// IO/CtrlInput
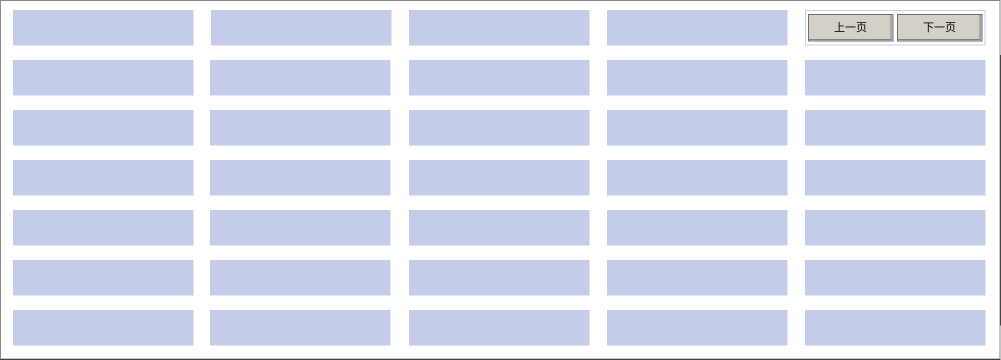
VISUALIZATION CtrlInput  // 1001x360
VAR_INPUT
	In:						POINTER TO BOOL;
	SizeIn:					DINT;
END_VAR
VAR
	_pageCount:				INT;
	_index:					INT;
END_VAR
    RoundedRectangle (0,0 1000x115)
    RoundedRectangle (0,245 1000x115)
    Rectangle (0,71 1000x240)
    Line (1000,55) (1000,325)
    Line (0,65) (0,312)
    RoundedRectangle (13,10 180x35), colour toggle: In[_index], invisible if: SizeIn<=_index, text list: 'InputText', text index: _index
    RoundedRectangle (211,10 180x35), colour toggle: In[1+_index], invisible if: SizeIn<= 1+_index, text list: 'InputText', text index: 1+_index
    RoundedRectangle (409,10 180x35), colour toggle: In[2+_index], invisible if: SizeIn<= 2+_index, text list: 'InputText', text index: 2+_index
    RoundedRectangle (607,10 180x35), colour toggle: In[3+_index], invisible if: SizeIn<=3+_index, text list: 'InputText', text index: 3+_index
    RoundedRectangle (805,10 180x35)
    Button (808,14 85x27), "上一页"
        OnMouseClick: execute {
            IF _index-34>=0 THEN
            	_index:=_index-34;
            END_IF
        }
    Button (897,14 85x27), "下一页"
        OnMouseClick: execute {
            IF SizeIn>_index+34 THEN
            	_index:=_index+34;
            END_IF
        }
    RoundedRectangle (13,60 180x35), colour toggle: In[_index+4], invisible if: SizeIn<=_index+4, text list: 'InputText', text index: _index+4
    RoundedRectangle (210,60 180x35), colour toggle: In[_index+5], invisible if: SizeIn<=_index+5, text list: 'InputText', text index: _index+5
    RoundedRectangle (409,60 180x35), colour toggle: In[_index+6], invisible if: SizeIn<=_index+6, text list: 'InputText', text index: _index+6
    RoundedRectangle (607,60 180x35), colour toggle: In[_index+7], invisible if: SizeIn<=_index+7, text list: 'InputText', text index: _index+7
    RoundedRectangle (805,60 180x35), colour toggle: In[_index+8], invisible if: SizeIn<=_index+8, text list: 'InputText', text index: _index+8
    RoundedRectangle (13,110 180x35), colour toggle: In[_index+9], invisible if: SizeIn<=_index+9, text list: 'InputText', text index: _index+9
    RoundedRectangle (210,110 180x35), colour toggle: In[_index+10], invisible if: SizeIn<=_index+10, text list: 'InputText', text index: _index+10
    RoundedRectangle (409,110 180x35), colour toggle: In[_index+11], invisible if: SizeIn<=_index+11, text list: 'InputText', text index: _index+11
    RoundedRectangle (607,110 180x35), colour toggle: In[_index+12], invisible if: SizeIn<=_index+12, text list: 'InputText', text index: _index+12
    RoundedRectangle (805,110 180x35), colour toggle: In[_index+13], invisible if: SizeIn<=_index+13, text list: 'InputText', text index: _index+13
    RoundedRectangle (13,160 180x35), colour toggle: In[_index+14], invisible if: SizeIn<=_index+14, text list: 'InputText', text index: _index+14
    RoundedRectangle (210,160 180x35), colour toggle: In[_index+15], invisible if: SizeIn<=_index+15, text list: 'InputText', text index: _index+15
    RoundedRectangle (409,160 180x35), colour toggle: In[_index+16], invisible if: SizeIn<=_index+16, text list: 'InputText', text index: _index+16
    RoundedRectangle (607,160 180x35), colour toggle: In[_index+17], invisible if: SizeIn<=_index+17, text list: 'InputText', text index: _index+17
    RoundedRectangle (805,160 180x35), colour toggle: In[_index+18], invisible if: SizeIn<=_index+18, text list: 'InputText', text index: _index+18
    RoundedRectangle (13,210 180x35), colour toggle: In[_index+19], invisible if: SizeIn<=_index+19, text list: 'InputText', text index: _index+19
    RoundedRectangle (210,210 180x35), colour toggle: In[_index+20], invisible if: SizeIn<=_index+20, text list: 'InputText', text index: _index+20
    RoundedRectangle (409,210 180x35), colour toggle: In[_index+21], invisible if: SizeIn<=_index+21, text list: 'InputText', text index: _index+21
    RoundedRectangle (607,210 180x35), colour toggle: In[_index+22], invisible if: SizeIn<=_index+22, text list: 'InputText', text index: _index+22
    RoundedRectangle (805,210 180x35), colour toggle: In[_index+23], invisible if: SizeIn<=_index+23, text list: 'InputText', text index: _index+23
    RoundedRectangle (13,260 180x35), colour toggle: In[_index+24], invisible if: SizeIn<=_index+24, text list: 'InputText', text index: _index+24
    RoundedRectangle (409,260 180x35), colour toggle: In[_index+26], invisible if: SizeIn<=_index+26, text list: 'InputText', text index: _index+26
    RoundedRectangle (210,260 180x35), colour toggle: In[_index+25], invisible if: SizeIn<=_index+25, text list: 'InputText', text index: _index+25
    RoundedRectangle (607,260 180x35), colour toggle: In[_index+27], invisible if: SizeIn<=_index+27, text list: 'InputText', text index: _index+27
    RoundedRectangle (805,260 180x35), colour toggle: In[_index+28], invisible if: SizeIn<=_index+28, text list: 'InputText', text index: _index+28
    RoundedRectangle (13,310 180x35), colour toggle: In[_index+29], invisible if: SizeIn<=_index+29, text list: 'InputText', text index: _index+29
    RoundedRectangle (210,310 180x35), colour toggle: In[_index+30], invisible if: SizeIn<=_index+30, text list: 'InputText', text index: _index+30
    RoundedRectangle (409,310 180x35), colour toggle: In[_index+31], invisible if: SizeIn<=_index+31, text list: 'InputText', text index: _index+31
    RoundedRectangle (607,310 180x35), colour toggle: In[_index+32], invisible if: SizeIn<=_index+32, text list: 'InputText', text index: _index+32
    RoundedRectangle (805,310 180x35), colour toggle: In[_index+33], invisible if: SizeIn<=_index+33, text list: 'InputText', text index: _index+33
END_VISUALIZATION

// IO/CtrlOutput
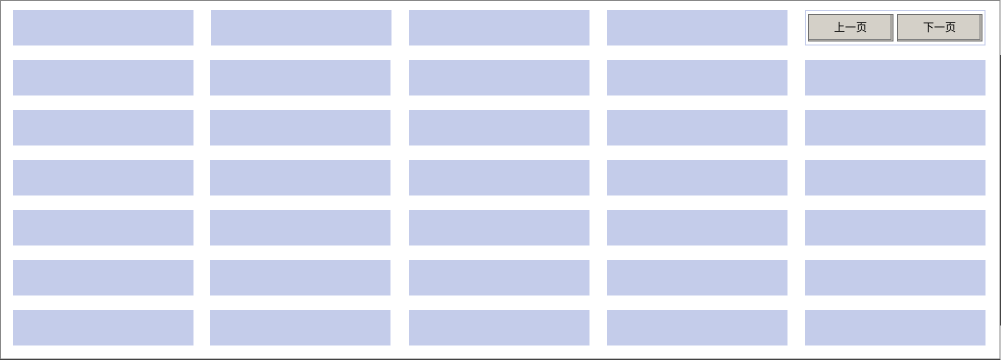
VISUALIZATION CtrlOutput  // 1001x360
VAR_INPUT
	In:						POINTER TO BOOL;
	SizeIn:					DINT;
	System:					REFERENCE TO ST_System;
END_VAR
VAR
	_pageCount:				INT;
	_index:					INT;
END_VAR
    RoundedRectangle (0,0 1000x115)
    RoundedRectangle (0,245 1000x115)
    Rectangle (0,71 1000x240)
    Line (1000,55) (1000,325)
    Line (0,65) (0,312)
    RoundedRectangle (13,10 180x35), colour toggle: In[_index], invisible if: SizeIn<=_index, text list: 'OutputText', text index: _index
        OnMouseClick: execute {
            IF System.stMode.bSetting AND SizeIn>_index THEN
            	In[_index]:=NOT In[_index];
            END_IF;
        }
    RoundedRectangle (211,10 180x35), colour toggle: In[1+_index], invisible if: SizeIn<= 1+_index, text list: 'OutputText', text index: 1+_index
        OnMouseClick: execute {
            IF System.stMode.bSetting AND SizeIn>_index+1 THEN
            	In[_index+1]:=NOT In[_index+1];
            END_IF;
        }
    RoundedRectangle (409,10 180x35), colour toggle: In[2+_index], invisible if: SizeIn<= 2+_index, text list: 'OutputText', text index: 2+_index
        OnMouseClick: execute {
            IF System.stMode.bSetting AND SizeIn>_index+2 THEN
            	In[_index+2]:=NOT In[_index+2];
            END_IF;
        }
    RoundedRectangle (607,10 180x35), colour toggle: In[3+_index], invisible if: SizeIn<=3+_index, text list: 'OutputText', text index: 3+_index
        OnMouseClick: execute {
            IF System.stMode.bSetting AND SizeIn>_index+3 THEN
            	In[_index+3]:=NOT In[_index+3];
            END_IF;
        }
    RoundedRectangle (805,10 180x35)
    RoundedRectangle (13,60 180x35), colour toggle: In[_index+4], invisible if: SizeIn<=_index+4, text list: 'OutputText', text index: _index+4
        OnMouseClick: execute {
            IF System.stMode.bSetting AND SizeIn>_index+4 THEN
            	In[_index+4]:=NOT In[_index+4];
            END_IF;
        }
    RoundedRectangle (210,60 180x35), colour toggle: In[_index+5], invisible if: SizeIn<=_index+5, text list: 'OutputText', text index: _index+5
        OnMouseClick: execute {
            IF System.stMode.bSetting AND SizeIn>_index+5 THEN
            	In[_index+5]:=NOT In[_index+5];
            END_IF;
        }
    RoundedRectangle (409,60 180x35), colour toggle: In[_index+6], invisible if: SizeIn<=_index+6, text list: 'OutputText', text index: _index+6
        OnMouseClick: execute {
            IF System.stMode.bSetting AND SizeIn>_index+6 THEN
            	In[_index+6]:=NOT In[_index+6];
            END_IF;
        }
    RoundedRectangle (607,60 180x35), colour toggle: In[_index+7], invisible if: SizeIn<=_index+7, text list: 'OutputText', text index: _index+7
        OnMouseClick: execute {
            IF System.stMode.bSetting AND SizeIn>_index+7 THEN
            	In[_index+7]:=NOT In[_index+7];
            END_IF;
        }
    RoundedRectangle (805,60 180x35), colour toggle: In[_index+8], invisible if: SizeIn<=_index+8, text list: 'OutputText', text index: _index+8
        OnMouseClick: execute {
            IF System.stMode.bSetting AND SizeIn>_index+8 THEN
            	In[_index+8]:=NOT In[_index+8];
            END_IF;
        }
    RoundedRectangle (13,110 180x35), colour toggle: In[_index+9], invisible if: SizeIn<=_index+9, text list: 'OutputText', text index: _index+9
        OnMouseClick: execute {
            IF System.stMode.bSetting AND SizeIn>_index+9 THEN
            	In[_index+9]:=NOT In[_index+9];
            END_IF;
        }
    RoundedRectangle (210,110 180x35), colour toggle: In[_index+10], invisible if: SizeIn<=_index+10, text list: 'OutputText', text index: _index+10
        OnMouseClick: execute {
            IF System.stMode.bSetting AND SizeIn>_index+10 THEN
            	In[_index+10]:=NOT In[_index+10];
            END_IF;
        }
    RoundedRectangle (409,110 180x35), colour toggle: In[_index+11], invisible if: SizeIn<=_index+11, text list: 'OutputText', text index: _index+11
        OnMouseClick: execute {
            IF System.stMode.bSetting AND SizeIn>_index+11 THEN
            	In[_index+11]:=NOT In[_index+11];
            END_IF;
        }
    RoundedRectangle (607,110 180x35), colour toggle: In[_index+12], invisible if: SizeIn<=_index+12, text list: 'OutputText', text index: _index+12
        OnMouseClick: execute {
            IF System.stMode.bSetting AND SizeIn>_index+12 THEN
            	In[_index+12]:=NOT In[_index+12];
            END_IF;
        }
    RoundedRectangle (805,110 180x35), colour toggle: In[_index+13], invisible if: SizeIn<=_index+13, text list: 'OutputText', text index: _index+13
        OnMouseClick: execute {
            IF System.stMode.bSetting AND SizeIn>_index+13 THEN
            	In[_index+13]:=NOT In[_index+13];
            END_IF;
        }
    RoundedRectangle (13,160 180x35), colour toggle: In[_index+14], invisible if: SizeIn<=_index+14, text list: 'OutputText', text index: _index+14
        OnMouseClick: execute {
            IF System.stMode.bSetting AND SizeIn>_index+14 THEN
            	In[_index+14]:=NOT In[_index+14];
            END_IF;
        }
    RoundedRectangle (210,160 180x35), colour toggle: In[_index+15], invisible if: SizeIn<=_index+15, text list: 'OutputText', text index: _index+15
        OnMouseClick: execute {
            IF System.stMode.bSetting AND SizeIn>_index+15 THEN
            	In[_index+15]:=NOT In[_index+15];
            END_IF;
        }
    RoundedRectangle (409,160 180x35), colour toggle: In[_index+16], invisible if: SizeIn<=_index+16, text list: 'OutputText', text index: _index+16
        OnMouseClick: execute {
            IF System.stMode.bSetting AND SizeIn>_index+16 THEN
            	In[_index+16]:=NOT In[_index+16];
            END_IF;
        }
    RoundedRectangle (607,160 180x35), colour toggle: In[_index+17], invisible if: SizeIn<=_index+17, text list: 'OutputText', text index: _index+17
        OnMouseClick: execute {
            IF System.stMode.bSetting AND SizeIn>_index+17 THEN
            	In[_index+17]:=NOT In[_index+17];
            END_IF;
        }
    RoundedRectangle (805,160 180x35), colour toggle: In[_index+18], invisible if: SizeIn<=_index+18, text list: 'OutputText', text index: _index+18
        OnMouseClick: execute {
            IF System.stMode.bSetting AND SizeIn>_index+18 THEN
            	In[_index+18]:=NOT In[_index+18];
            END_IF;
        }
    RoundedRectangle (13,210 180x35), colour toggle: In[_index+19], invisible if: SizeIn<=_index+19, text list: 'OutputText', text index: _index+19
        OnMouseClick: execute {
            IF System.stMode.bSetting AND SizeIn>_index+19 THEN
            	In[_index+19]:=NOT In[_index+19];
            END_IF;
        }
    RoundedRectangle (210,210 180x35), colour toggle: In[_index+20], invisible if: SizeIn<=_index+20, text list: 'OutputText', text index: _index+20
        OnMouseClick: execute {
            IF System.stMode.bSetting AND SizeIn>_index+20 THEN
            	In[_index+20]:=NOT In[_index+20];
            END_IF;
        }
    RoundedRectangle (409,210 180x35), colour toggle: In[_index+21], invisible if: SizeIn<=_index+21, text list: 'OutputText', text index: _index+21
        OnMouseClick: execute {
            IF System.stMode.bSetting AND SizeIn>_index+21 THEN
            	In[_index+21]:=NOT In[_index+21];
            END_IF;
        }
    RoundedRectangle (607,210 180x35), colour toggle: In[_index+22], invisible if: SizeIn<=_index+22, text list: 'OutputText', text index: _index+22
        OnMouseClick: execute {
            IF System.stMode.bSetting AND SizeIn>_index+22 THEN
            	In[_index+22]:=NOT In[_index+22];
            END_IF;
        }
    RoundedRectangle (805,210 180x35), colour toggle: In[_index+23], invisible if: SizeIn<=_index+23, text list: 'OutputText', text index: _index+23
        OnMouseClick: execute {
            IF System.stMode.bSetting AND SizeIn>_index+23 THEN
            	In[_index+23]:=NOT In[_index+23];
            END_IF;
        }
    RoundedRectangle (13,260 180x35), colour toggle: In[_index+24], invisible if: SizeIn<=_index+24, text list: 'OutputText', text index: _index+24
        OnMouseClick: execute {
            IF System.stMode.bSetting AND SizeIn>_index+24 THEN
            	In[_index+24]:=NOT In[_index+24];
            END_IF;
        }
    RoundedRectangle (409,260 180x35), colour toggle: In[_index+26], invisible if: SizeIn<=_index+26, text list: 'OutputText', text index: _index+26
        OnMouseClick: execute {
            IF System.stMode.bSetting AND SizeIn>_index+26 THEN
            	In[_index+26]:=NOT In[_index+26];
            END_IF;
        }
    RoundedRectangle (210,260 180x35), colour toggle: In[_index+25], invisible if: SizeIn<=_index+25, text list: 'OutputText', text index: _index+25
        OnMouseClick: execute {
            IF System.stMode.bSetting AND SizeIn>_index+25 THEN
            	In[_index+25]:=NOT In[_index+25];
            END_IF;
        }
    RoundedRectangle (607,260 180x35), colour toggle: In[_index+27], invisible if: SizeIn<=_index+27, text list: 'OutputText', text index: _index+27
        OnMouseClick: execute {
            IF System.stMode.bSetting AND SizeIn>_index+27 THEN
            	In[_index+27]:=NOT In[_index+27];
            END_IF;
        }
    RoundedRectangle (805,260 180x35), colour toggle: In[_index+28], invisible if: SizeIn<=_index+28, text list: 'OutputText', text index: _index+28
        OnMouseClick: execute {
            IF System.stMode.bSetting AND SizeIn>_index+28 THEN
            	In[_index+28]:=NOT In[_index+28];
            END_IF;
        }
    RoundedRectangle (13,310 180x35), colour toggle: In[_index+29], invisible if: SizeIn<=_index+29, text list: 'OutputText', text index: _index+29
        OnMouseClick: execute {
            IF System.stMode.bSetting AND SizeIn>_index+29 THEN
            	In[_index+29]:=NOT In[_index+29];
            END_IF;
        }
    RoundedRectangle (210,310 180x35), colour toggle: In[_index+30], invisible if: SizeIn<=_index+30, text list: 'OutputText', text index: _index+30
        OnMouseClick: execute {
            IF System.stMode.bSetting AND SizeIn>_index+30 THEN
            	In[_index+30]:=NOT In[_index+30];
            END_IF;
        }
    RoundedRectangle (409,310 180x35), colour toggle: In[_index+31], invisible if: SizeIn<=_index+31, text list: 'OutputText', text index: _index+31
        OnMouseClick: execute {
            IF System.stMode.bSetting AND SizeIn>_index+31 THEN
            	In[_index+31]:=NOT In[_index+31];
            END_IF;
        }
    RoundedRectangle (607,310 180x35), colour toggle: In[_index+32], invisible if: SizeIn<=_index+32, text list: 'OutputText', text index: _index+32
        OnMouseClick: execute {
            IF System.stMode.bSetting AND SizeIn>_index+32 THEN
            	In[_index+32]:=NOT In[_index+32];
            END_IF;
        }
    RoundedRectangle (805,310 180x35), colour toggle: In[_index+33], invisible if: SizeIn<=_index+33, text list: 'OutputText', text index: _index+33
        OnMouseClick: execute {
            IF System.stMode.bSetting AND SizeIn>_index+33 THEN
            	In[_index+33]:=NOT In[_index+33];
            END_IF;
        }
    Button (897,14 85x27), "下一页"
        OnMouseClick: execute {
            IF SizeIn>_index+34 THEN
            	_index:=_index+34;
            END_IF
        }
    Button (808,14 85x27), "上一页"
        OnMouseClick: execute {
            IF _index-34>=0 THEN
            	_index:=_index-34;
            END_IF
        }
END_VISUALIZATION

// Recipe/VISUs/CtrlRecipe
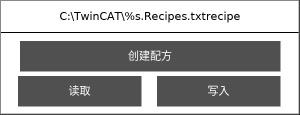
VISUALIZATION CtrlRecipe  // 300x115
    RoundedRectangle (0,0 300x115)
    Rectangle (5,4 290x25), "C:\TwinCAT\%s.Recipes.txtrecipe", text variable: P_Recipe._sRecipeName
        OnMouseClick: write the text variable via Edit
    Line (0,32) (300,32)
    RoundedRectangle (20,41 260x30), "创建配方", input disabled if: P_Recipe._bLock
        tap P_Recipe._bRecipeCreate
    RoundedRectangle (18,76 123x30), "读取", input disabled if: P_Recipe._bLock
        tap P_Recipe._bRecipeRead
    RoundedRectangle (157,76 123x30), "写入", input disabled if: P_Recipe._bLock
        tap P_Recipe._bRecipeWrite
END_VISUALIZATION

// System/VISUs/CtrlAxisCylinder
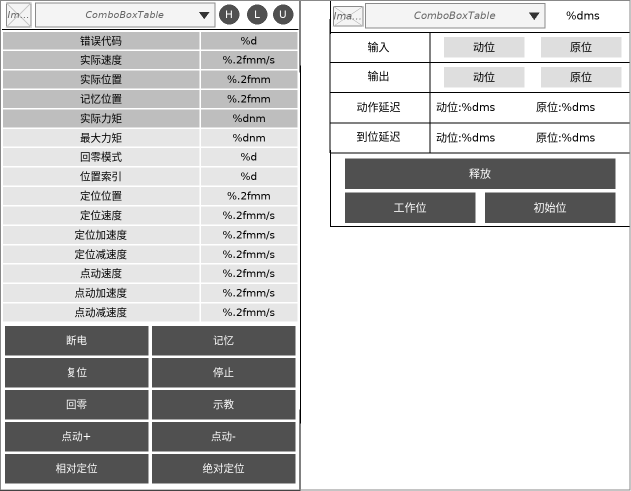
VISUALIZATION CtrlAxisCylinder  // 631x491
    Frame (0,0 301x491)
        shows CtrlAxisGroup(System := G_stSystem, Axis := G_arrAxis, Data := G_arrAxisData)
    Frame (330,0 301x227)
        shows CtrlCylinderGroup(System := G_stSystem, Cylinder := G_arrCylinder, CylinderData := G_arrCylinderData)
END_VISUALIZATION

// System/VISUs/CtrlBtnBox
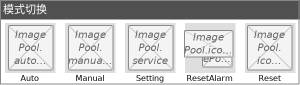
VISUALIZATION CtrlBtnBox  // 300x85
VAR_INPUT
	System:						REFERENCE TO ST_System;
END_VAR
    Rectangle (0,20 300x65)
    RoundedRectangle (5,23 50x50), colour toggle: System.stMode.bAuto
    Image (8,25 45x45), image: ImagePool.auto_mode_80x80
        OnMouseDown: execute { System.stInput.bAuto:=true; }
        OnMouseUp: execute { System.stInput.bAuto:=false; }
    Rectangle (0,0 300x19), "模式切换"
    RoundedRectangle (65,23 50x50), colour toggle: System.stMode.bManual
    Image (68,25 45x45), image: ImagePool.manual_mode_80x80
        OnMouseDown: execute { System.stInput.bManual:=true; }
        OnMouseUp: execute { System.stInput.bManual:=false; }
    RoundedRectangle (125,23 50x50), colour toggle: System.stMode.bSetting
    Image (128,25 45x45), image: ImagePool.service
        OnMouseDown: execute { System.stInput.bSetting:=true; }
        OnMouseUp: execute { System.stInput.bSetting:=false; }
    RoundedRectangle (185,23 50x50), colour toggle: System.stMode.bAlarming
    RoundedRectangle (245,23 50x50), colour toggle: System.stInput.bReset
    Image (247,25 45x45), image: ImagePool.ico_version_history
        OnMouseDown: execute { System.stInput.bReset:=true; }
        OnMouseUp: execute { System.stInput.bReset:=false; }
    Image (202,37 30x30), image: ImagePool.ico_menu_alarm
    Image (184,30 49x27), image: ImagePool.ico_menu_clean
        OnMouseDown: execute { System.stInput.bResetAlarm:=true; }
        OnMouseUp: execute { System.stInput.bResetAlarm:=false; }
    Rectangle (5,73 50x11), "Auto"
    Rectangle (65,73 50x11), "Manual"
    Rectangle (125,73 50x11), "Setting"
    Rectangle (185,73 50x11), "ResetAlarm"
    Rectangle (245,73 50x11), "Reset"
END_VISUALIZATION

// System/VISUs/CtrlBtnLogin
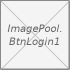
VISUALIZATION CtrlBtnLogin  // 70x70
    Image (0,0 70x70), image: ImagePool.BtnLogin1
        OnMouseClick:  Type=Login
END_VISUALIZATION

// System/VISUs/CtrlFormColse
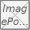
VISUALIZATION CtrlFormColse  // 30x30
    Image (0,0 30x30), image: ImagePool.cross-512
        OnMouseClick:  ExecuteCommand=ExecuteCommand=[Command=ExecuteClientProgram, Value='TaskKILL/IM', Value2='Tc3PlcHmi.exe']
END_VISUALIZATION

// System/VISUs/CtrlHomeGroup
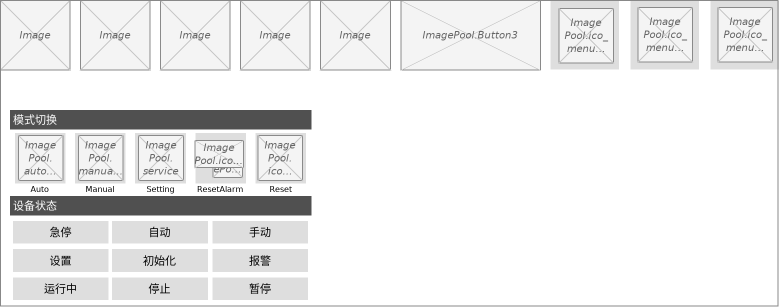
VISUALIZATION CtrlHomeGroup  // 779x307
    Frame (0,0 779x70)
        shows CtrlPageSwitch(System := G_stSystem)
    Frame (10,110 301x86)
        shows CtrlBtnBox(System := G_stSystem)
    Frame (10,196 301x111)
        shows CtrlMode(System := G_stSystem)
END_VISUALIZATION

// System/VISUs/CtrlLanguage
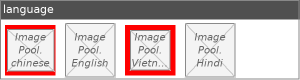
VISUALIZATION CtrlLanguage  // 300x80
VAR_INPUT
	System:					REFERENCE TO ST_System;
END_VAR
    Rectangle (0,20 300x60)
    Rectangle (0,0 300x19), "language"
    RoundedRectangle (5,25 50x50)
    Image (7,29 47x42), image: ImagePool.chinese
        OnMouseClick:  ChangeLanguage=Chinese
        OnMouseClick: execute { system.stMode.eLanguage:=E_Language.Chinese; }
    Image (65,23 50x54), image: ImagePool.English
        OnMouseClick:  ChangeLanguage=English
        OnMouseClick: execute { system.stMode.eLanguage:=E_Language.English; }
    RoundedRectangle (125,25 50x50)
        OnMouseClick:  ChangeLanguage=Vietnamese
    Image (130,30 40x40), image: ImagePool.Vietnamese
        OnMouseClick:  ChangeLanguage=Vietnamese
        OnMouseClick: execute { system.stMode.eLanguage:=E_Language.Vietnamese; }
    Image (185,23 50x54), image: ImagePool.Hindi
        OnMouseClick:  ChangeLanguage=Hindi
        OnMouseClick: execute { system.stMode.eLanguage:=E_Language.Hindi; }
END_VISUALIZATION

// System/VISUs/CtrlMode
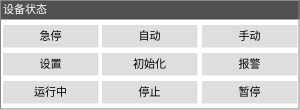
VISUALIZATION CtrlMode  // 300x110
VAR_INPUT
	System:					REFERENCE TO ST_System;
END_VAR
    Rectangle (0,20 300x90)
    Rectangle (0,0 300x19), "设备状态"
    RoundedRectangle (3,25 95x22), "急停", colour toggle: System.stMode.bEStop
    RoundedRectangle (102,25 95x22), "自动", colour toggle: system.stMode.bAuto
    RoundedRectangle (202,25 95x22), "手动", colour toggle: System.stMode.bManual
    RoundedRectangle (3,53 95x22), "设置", colour toggle: System.stMode.bSetting
    RoundedRectangle (3,81 95x22), "运行中", colour toggle: System.stMode.bAutoRunning
    RoundedRectangle (102,53 95x22), "初始化", colour toggle: System.stMode.bHoming
    RoundedRectangle (102,81 95x22), "停止", colour toggle: System.stMode.bStop
    RoundedRectangle (202,81 95x22), "暂停", colour toggle: System.stMode.bPause
    RoundedRectangle (202,53 95x22), "报警", colour toggle: System.stMode.bAlarming
END_VISUALIZATION

// System/VISUs/CtrlPageSwitch
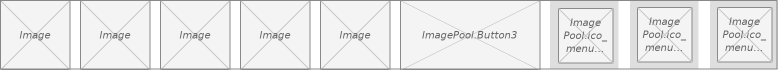
VISUALIZATION CtrlPageSwitch  // 778x70
VAR_INPUT// PageHome,PageSetting,PageMonitor,PageMessage,PageData
	System:				REFERENCE TO ST_System;
END_VAR
    ImageSwitcher (0,0 70x70), variable: System.iPageNow=0, background image: ImagePool.BtnHome2, image: ImagePool.BtnHome1, behaviour: TOGGLE
    ImageSwitcher (320,0 70x70), variable: System.iPageNow=40, background image: ImagePool.BtnData2, image: ImagePool.BtnData1, behaviour: TOGGLE
    ImageSwitcher (80,0 70x70), variable: System.iPageNow=10, background image: ImagePool.BtnSetting1, image: ImagePool.BtnSetting2, behaviour: TOGGLE
    ImageSwitcher (160,0 70x70), variable: System.iPageNow=20, background image: ImagePool.IO2, image: ImagePool.IO1, behaviour: TOGGLE
    ImageSwitcher (240,0 70x70), variable: System.iPageNow=30, background image: ImagePool.BtnInfo2, image: ImagePool.BtnInfo1, behaviour: TOGGLE
    Image (0,0 70x70)
        OnMouseClick:  Assign=PageHome, Type=Assignment
        OnMouseClick: execute { System.iPageNow:=0; }
    Image (320,0 70x70)
        OnMouseClick:  Assign=PageData, Type=Assignment
        OnMouseClick: execute { System.iPageNow:=40; }
    Image (80,0 70x70)
        OnMouseClick:  Assign=PageSetting, Type=Assignment
        OnMouseClick: execute { System.iPageNow:=10; }
    Image (240,0 70x70)
        OnMouseClick:  Assign=PageMessage, Type=Assignment
        OnMouseClick: execute { System.iPageNow:=30; }
    Image (160,0 70x70)
        OnMouseClick:  Assign=PageMonitor, Type=Assignment
        OnMouseClick: execute { System.iPageNow:=20; }
    Image (400,0 140x70), image: ImagePool.Button3
    RoundedRectangle (550,1 68x68), colour toggle: System.stMode.bAutoRunning OR System.stMode.bHoming
    Image (558,8 55x55), image: ImagePool.ico_menu_play
        OnMouseDown: execute { System.stInput.bStart:=true; }
        OnMouseUp: execute { System.stInput.bStart:=false; }
    RoundedRectangle (630,1 68x68), colour toggle: System.stMode.bStop
    RoundedRectangle (710,1 68x68), colour toggle: System.stMode.bPause
    Image (637,7 55x55), image: ImagePool.ico_menu_pause
        OnMouseDown: execute { System.stInput.bStop:=true; }
        OnMouseUp: execute { System.stInput.bStop:=false; }
    Image (717,7 55x55), image: ImagePool.ico_menu_stop
        OnMouseDown: execute { System.stInput.bPause:=true; }
        OnMouseUp: execute { System.stInput.bPause:=false; }
END_VISUALIZATION

// System/VISUs/CtrlStation
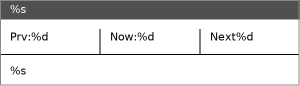
VISUALIZATION CtrlStation  // 300x86
VAR_INPUT
	System:					REFERENCE TO ST_System;
	Station:				REFERENCE TO ST_SystemStation;
END_VAR
    Rectangle (0,0 300x86)
    Rectangle (0,0 300x19), "%s", text variable: Station.arrName[System.stMode.eLanguage]
    Rectangle (0,22 100x30), "Prv:%d", text variable: Station.iStepPrev
    Rectangle (100,22 100x30), "Now:%d", text variable: Station.iStepNow
    Rectangle (200,22 100x30), "Next%d", text variable: Station.iStepNext
    Rectangle (0,56 300x30), "%s", text variable: Station.arrInfo[System.stMode.eLanguage]
    Line (100,54) (100,29)
    Line (200,54) (200,29)
    Line (1,54) (299,54)
END_VISUALIZATION

// TcpIp/VISUs/CtrlTcpIpClient
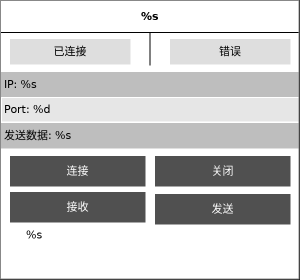
VISUALIZATION CtrlTcpIpClient  // 300x280
VAR_IN_OUT
	TcpIpClient:					ST_TcpIpClient;
	Data:							ST_TcpIpData;
END_VAR
    RoundedRectangle (0,0 300x280)
    Rectangle (25,4 250x25), "%s", text variable: TcpIpClient.sName
    Rectangle (23,227 255x48), "%s", text variable: TcpIpClient.sReceiveData
    Line (0,32) (300,32)
    RoundedRectangle (10,39 120x25), "已连接", colour toggle: TcpIpClient.stStatus.bConnected
    RoundedRectangle (170,39 120x25), "错误", colour toggle: TcpIpClient.stStatus.bError
    Rectangle (1,72 298x25), "IP: %s", text variable: Data.sServerIp
        OnMouseDown: write the text variable via VisuDialogs.Numpad
    Rectangle (1,97 298x25), "Port: %d", text variable: Data.iServerPort
        OnMouseDown: write the text variable via VisuDialogs.Numpad
    Rectangle (1,123 298x25), "发送数据: %s", text variable: TcpIpClient.sSendData
        OnMouseDown: write the text variable via Default
    Line (150,65) (150,32)
    RoundedRectangle (10,156 135x30), "连接", input disabled if: TcpIpClient.stStatus.bConnecting
        tap TcpIpClient.stContorl.stConnect.bManual
    RoundedRectangle (155,156 135x30), "关闭", input disabled if: TcpIpClient.stStatus.bClosing
        tap TcpIpClient.stContorl.stClose.bManual
    RoundedRectangle (10,192 135x30), "接收"
        tap TcpIpClient.stContorl.stReceive.bManual
    RoundedRectangle (155,194 135x30), "发送", input disabled if: TcpIpClient.stStatus.bSending
        tap TcpIpClient.stContorl.stSend.bManual
END_VISUALIZATION

// Yield/VISUs/CtrlYield
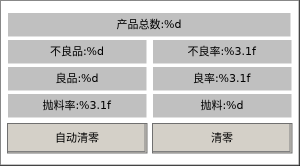
VISUALIZATION CtrlYield  // 300x166
VAR_INPUT
	Yield:					REFERENCE TO ST_Yield;
	Data:					REFERENCE TO ST_YieldData;
END_VAR
    RoundedRectangle (0,0 300x166)
    Rectangle (7,12 284x25), "产品总数:%d", text variable: Data.iAll
    Button (152,123 140x30), "清零"
        tap Yield.stControl.bClear
    Rectangle (7,66 140x25), "良品:%d", text variable: Data.iOK
    Rectangle (7,39 140x25), "不良品:%d", text variable: Data.iNG
    Rectangle (152,66 140x25), "良率:%3.1f", text variable: Data.fOkPercentage
    Rectangle (152,39 140x25), "不良率:%3.1f", text variable: Data.fNgPercentage
    Rectangle (152,93 140x25), "抛料:%d", text variable: Data.iTOSS
    Button (7,123 140x30), "自动清零"
        toggle Yield.stControl.bAutoClear p2164770859=TRUE
    Rectangle (7,93 140x25), "抛料率:%3.1f", text variable: Data.fTOSSPercentage
END_VISUALIZATION

(* text list TextHomeMode (id | default | Chinese | English | Vietnamese | Hindi)
  0 | 原点信号 | 原点信号 | Bool | là gì | बूल
  1 | 扭矩信号 | 扭矩信号 | Torque | Mô-men xoắn | घूर्णन-बल
  2 | 当前位置 | 当前位置 | Direct | Trực tiếp | प्रत्यक्ष
  3 | 速度信号 | 速度信号 | Velocity | Vận tốc | वेग
   |  |  |  |  |  *)

(* text list InputText (id | default)
   |  *)

(* text list OutputText (id | default)
   |  *)
